TYPE ST_EM_Cfg :
	STRUCT
		CamActivationMode : INT;
	END_STRUCT
END_TYPE

(* stored: Version 1.1.0.1, ProductVersion 3.1.4024.12
   DUT ST_EM_Cfg: Id {121940d2-7b10-4ae7-9745-d573e2d834e3} *)
